FUNCTION_BLOCK RunUnitDummy EXTENDS RunUnitSlave
VAR_INPUT
END_VAR
VAR_OUTPUT
END_VAR
VAR
END_VAR
VAR PERSISTENT
	var1 : INT := 1;
	var2 : INT := 2;
END_VAR

METHOD ConfigureRead : CellDataBlock
VAR_INPUT
	input : CellDataBlock;
	mode : eModes;
END_VAR
//ConfigureRead := input;
CASE input.unit.config.configId OF
	0:
		 ConfigureRead.unit.config.value := TO_WORD(var1);
	1:
		ConfigureRead.unit.config.value := TO_WORD(var2);
END_CASE
END_METHOD

METHOD ConfigureWrite : BOOL
VAR_INPUT
	input : CellDataBlock;
	mode : eModes;
END_VAR
CASE input.unit.config.configId OF
	0:
		var1 := TO_INT(input.unit.config.value);
	1:
		var2 := TO_INT(input.unit.config.value);
END_CASE
END_METHOD

END_FUNCTION_BLOCK

(* stored: Version 1.1.0.1, ProductVersion 3.1.4022.10
   POU RunUnitDummy: Id {16212f14-bd08-4821-a28c-98ec1bf24c8e}, SpecialFunc None
   Method ConfigureRead: Id {b15ff683-22c9-407a-8a1a-145273f95434}
   Method ConfigureWrite: Id {9ea82dfa-8ca4-430d-9b3f-9d91ac6179f9} *)
